// TIA Portal V17 export
// export: Created 2024-09-02T12:50:34.8349517Z, ExportSetting WithDefaults, DisplayName Totally Integrated Automation Portal, DisplayVersion V17, DisplayName TIA Portal Openness, DisplayVersion V17, DisplayName TIA Portal Version Control Interface, DisplayVersion V17, DisplayName STEP 7 Professional, DisplayVersion V17, DisplayName STEP 7 Safety, DisplayVersion V17, DisplayName WinCC Professional, DisplayVersion V17
TYPE "typ_Einzelmeldung"
// stored: IsFailsafeCompliant false
   STRUCT
      meldung_byte_1 : Byte;   // Meldungsbit / message bit
      meldung_byte_2 : Byte;   // Meldungsbit / message bit
      meldung_byte_3 : Byte;   // Meldungsbit / message bit
      meldung_byte_4 : Byte;   // Meldungsbit / message bit
   END_STRUCT;
END_TYPE
